// TwinCAT 3 PLC project PLC
// ProgramVersion: 3.1.4024.0
// libraries:
//   Tc2_Standard, * (Beckhoff Automation GmbH)
//   Tc2_System, * (Beckhoff Automation GmbH)
//   Tc3_Module, * (Beckhoff Automation GmbH)
// project tree:
//   50_CONTROL_MODULE/00_COMMON/ E_ModuleState.TcDUT, ST_MODULE_ALARM.TcDUT
//   50_CONTROL_MODULE/10_VALVE/ E_ValveState.TcDUT, FB_Valve.TcPOU, ST_ValveConfig.TcDUT, ST_ValveData.TcDUT
//   / PlcTask.TcTTO (not stored)
//   POUs/ MAIN.TcPOU
// real-time tasks:
//   TASK PlcTask: cycle T#10ms, priority 20, ADS port 350

// ---- 50_CONTROL_MODULE/00_COMMON/E_ModuleState.TcDUT
{attribute 'qualified_only'}
{attribute 'strict'}
TYPE E_ModuleState :
(
    MANUAL := 0,   (* Manual mode *)
    AUTO := 1      (* Auto mode *)
);
END_TYPE;

// ---- 50_CONTROL_MODULE/00_COMMON/ST_MODULE_ALARM.TcDUT
TYPE ST_MODULE_ALARM :
STRUCT
	active		: BOOL;
	description	: STRING;
END_STRUCT
END_TYPE

// ---- 50_CONTROL_MODULE/10_VALVE/E_ValveState.TcDUT
{attribute 'qualified_only'}
{attribute 'strict'}
TYPE E_ValveState :
(
    VALVE_OFF := 0,
    VALVE_OPENING := 1,
    VALVE_OPEN := 2,
    VALVE_CLOSING := 3,
    VALVE_CLOSED := 4,
    VALVE_FAULT := 5
);
 END_TYPE;

// ---- 50_CONTROL_MODULE/10_VALVE/ST_ValveConfig.TcDUT
{attribute 'OPC.UA.DA' := '1'}
{attribute 'OPC.UA.DA.StructuredType' := '1'}
{attribute 'Retain' := 'True'}
TYPE ST_ValveConfig :
STRUCT
    tOpenTimeout   			: TIME := T#10S;        (* Timeout for opening the valve *)
    tCloseTimeout  			: TIME := T#10S;        (* Timeout for closing the valve *)
    bEnableOpenFeedback   	: BOOL := FALSE; (* Enable feedback for open status *)
    bEnableCloseFeedback  	: BOOL := FALSE; (* Enable feedback for close status *)
END_STRUCT
END_TYPE

// ---- 50_CONTROL_MODULE/10_VALVE/ST_ValveData.TcDUT
{attribute 'OPC.UA.DA' := '1'}
{attribute 'OPC.UA.DA.StructuredType' := '1'}
TYPE ST_ValveData :
STRUCT
    eState         	: E_ValveState;        (* Current state of the valve *)
	eModuleState   	: E_ModuleState;       (* Module state: Manual or Auto *)
    bEnabled       	: BOOL;                 (* Valve enable/disable status *)
    fault			: ST_MODULE_ALARM;		
    tElapsedTime   	: TIME;                 (* Time elapsed in current state *)
    lastOpenTime   	: TIME;                 (* Last time the valve spent opening *)
    lastCloseTime  	: TIME;                 (* Last time the valve spent closing *)
END_STRUCT
END_TYPE

// ---- 50_CONTROL_MODULE/10_VALVE/FB_Valve.TcPOU
FUNCTION_BLOCK FB_Valve
VAR_INPUT
    bEnable        		: BOOL;                 (* Enable valve control *)
    bAuto          		: BOOL;                 (* TRUE = Auto mode, FALSE = Manual mode *)
	b_InOpenFeedback	:BOOL;
	b_InCloseFeedback	:BOOL;	
END_VAR

VAR_OUTPUT
    b_OutOpenCommand   	:  BOOL;  
	b_OutCloseCommand   :  BOOL;       
END_VAR

VAR
	data 		   			: ST_ValveData  ;
	{attribute 'OPC.UA.DA' := '1'}
	{attribute 'OPC.UA.DA.StructuredType' := '1'}
	bManualOpen    			: BOOL;                 (* Manual open command *)
	{attribute 'OPC.UA.DA' := '1'}
	{attribute 'OPC.UA.DA.StructuredType' := '1'}
    bManualClose   			: BOOL;                 (* Manual close command *)
	{attribute 'OPC.UA.DA' := '1'}
	{attribute 'OPC.UA.DA.StructuredType' := '1'}
    bManualReset   			: BOOL;                 (* Manual reset command *)
    ton_MovementTime   		: TON;                	(* Timer for monitor current operation *)
	bStartMovement			: BOOL;
	bOutOpen				: BOOL;
	bOutClose				: BOOL;
END_VAR

VAR PERSISTENT
	stConfig       : ST_ValveConfig;      (* Valve configuration parameters *)
END_VAR

(* Module State logic *)
IF NOT bEnable THEN
    (* Valve is disabled - reset to OFF state *)
	M_PrivateOff();
    RETURN;
ELSIF bAuto THEN 
	data.eModuleState := E_ModuleState.AUTO;
ELSE
	data.eModuleState := E_ModuleState.MANUAL;
	M_PrivateManualMode();
END_IF


(* Main state handling *)
CASE data.eState OF		
    E_ValveState.VALVE_OPENING:

        IF ton_MovementTime.et >= stConfig.tOpenTimeout THEN
            (* Timeout occurred *)
            data.eState:= E_ValveState.VALVE_FAULT;
            data.fault.active := TRUE;
            data.fault.description := 'opening timeout';
        ELSIF b_InOpenFeedback AND stConfig.bEnableOpenFeedback THEN
           	data.eState:= E_ValveState.VALVE_OPEN;
			data.lastOpenTime := ton_MovementTime.PT ;
			bStartMovement := FALSE;
		ELSIF NOT stConfig.bEnableOpenFeedback THEN
			data.eState:= E_ValveState.VALVE_OPEN;
			bStartMovement := FALSE;
        END_IF

	E_ValveState.VALVE_CLOSING:
        IF ton_MovementTime.et >= stConfig.tCloseTimeout THEN
            (* Timeout occurred *)
            data.eState:= E_ValveState.VALVE_FAULT;
            data.fault.active := TRUE;
            data.fault.description := 'closing timeout';
        ELSIF b_InCloseFeedback AND stConfig.bEnableCloseFeedback THEN
           	data.eState:= E_ValveState.VALVE_CLOSED;
			data.lastOpenTime := ton_MovementTime.PT ;
			bStartMovement := FALSE;
		ELSIF NOT stConfig.bEnableOpenFeedback THEN
			data.eState:= E_ValveState.VALVE_CLOSED;
			bStartMovement := FALSE;
        END_IF

    E_ValveState.VALVE_FAULT:
        (* Fault Handling: Manual reset or auto-clear can be added here *)
        (* In this simple example, it remains in fault state until reset manually *)
	

END_CASE;

ton_MovementTime(IN:=bStartMovement, PT:=T#2147483647MS );

METHOD closeAuto : BOOL
IF data.eModuleState = E_ModuleState.AUTO THEN
	M_PrivateCloseValve();
END_IF
END_METHOD

METHOD PRIVATE M_PrivateCloseValve : BOOL
data.eState := E_ValveState.VALVE_CLOSING;
data.lastCloseTime := T#0S;  (* Reset last open time *)
bStartMovement := TRUE;
data.tElapsedTime := T#0S;
bOutOpen := FALSE;
bOutClose:= TRUE;
END_METHOD

METHOD PRIVATE M_PrivateManualMode : BOOL
IF data.eModuleState = E_ModuleState.MANUAL THEN
	IF bManualOpen THEN 
		bManualOpen := FALSE;
		M_PrivateOpenValve();
	ELSIF bManualClose THEN 
		bManualClose := FALSE;
		M_PrivateCloseValve();
	ELSIF bManualReset THEN 
		bManualReset := FALSE;
		M_resetFault();
	END_IF
END_IF
END_METHOD

METHOD PRIVATE M_PrivateOff : BOOL
data.eState := E_ValveState.VALVE_OFF;
data.lastOpenTime := T#0S;  (* Reset last open time *)
data.tElapsedTime := T#0S;
bOutOpen := FALSE;
bOutClose:= FALSE;
M_resetFault();
END_METHOD

METHOD PRIVATE M_PrivateOpenValve : BOOL
data.eState := E_ValveState.VALVE_OPENING;
data.lastOpenTime := T#0S;  (* Reset last open time *)
bStartMovement := TRUE;
data.tElapsedTime := T#0S;
bOutOpen := TRUE;
bOutClose:= FALSE;
END_METHOD

METHOD M_resetFault : BOOL
data.fault.active := FALSE;
data.fault.description := '';
data.eState := E_ValveState.VALVE_OFF;
END_METHOD

METHOD openAuto : BOOL
IF data.eModuleState = E_ModuleState.AUTO THEN
	M_PrivateOpenValve();
END_IF
END_METHOD

END_FUNCTION_BLOCK

// ---- POUs/MAIN.TcPOU
PROGRAM MAIN
VAR
	valve1			: FB_Valve;
END_VAR

valve1(bEnable:=TRUE );

END_PROGRAM
